FUNCTION_BLOCK AssemblySequenceStop EXTENDS AssemblySequence IMPLEMENTS ZCore.ISequence
VAR
  _step : ZCore.Step(AssemblyStep.StopBegin, AssemblyStep.StopEnd);
  _timerSim : ZAux.Timer;
END_VAR

IF OnStart(_step) THEN
  ; // init custom sequence variables here ...
END_IF

REPEAT
  LogStep();

  CASE _step.Index OF
    (* -------------------------------------------------------------------------------------------------------------------------------- *)
    AssemblyStep.StopBegin:
    (* -------------------------------------------------------------------------------------------------------------------------------- *)
      IF _step.OnEntry()
      THEN
        _timerSim.WaitAsync(5);
			END_IF
      
      Await(_timerSim, nextStep:=AssemblyStep.StopEnd);
      // _step.SetNext(index:=AssemblyStep.StopEnd);

    (* -------------------------------------------------------------------------------------------------------------------------------- *)
    AssemblyStep.StopEnd:
    (* -------------------------------------------------------------------------------------------------------------------------------- *)    
      SetBusy(FALSE);
  
  ELSE
    Abort('sequence contains unhandled step');
  END_CASE
UNTIL _step.IsNotRepeatable() OR_ELSE NOT Busy END_REPEAT

END_FUNCTION_BLOCK

(* stored: Version 1.1.0.1
   POU AssemblySequenceStop: Id {61bb870f-faec-4e05-894b-34850fd75560}, SpecialFunc None *)
